{attribute 'qualified_only'}
VAR_GLOBAL
	UnitPackTags : ARRAY [1..5] OF ST_PackMLv30Ext ;
	LineCommands : ST_PackMLv30Ext;
END_VAR

(* stored: Version 1.1.0.1, ProductVersion 3.1.4024.11
   GVL GVL: Id {2bb718b5-10f5-4e26-99ca-be5abeecc303} *)
